TYPE ST_Field :
STRUCT
	FieldName			: STRING(255);
	FieldValue			: STRING(255);
END_STRUCT
END_TYPE

(* stored: Version 1.1.0.1, ProductVersion 3.1.4024.11
   DUT ST_Field: Id {3716c8ee-a72e-4952-8c4b-c162e8428f7a} *)
